TYPE ST_Task_Info :
STRUCT
	sName			: STRING;
	rCycleTime		: REAL;
	rLastExecTime	: REAL;
	rPercentUsage	: REAL;
	iExceedCounter	: DINT;
	bResetCounter	: BOOL;
END_STRUCT
END_TYPE

(* stored: Version 1.1.0.1, ProductVersion 3.1.4024.0
   DUT ST_Task_Info: Id {b60342db-3e35-44cf-9ad1-2ed8bbce7665} *)
